// TwinCAT 3 PLC project Untitled1
// ProgramVersion: 3.1.4023.0
// libraries:
//   Motion, * (Ljmu)
//   SafetyMonitoring, * (Ljmu)
//   Tc2_ControllerToolbox, * (Beckhoff Automation GmbH)
//   Tc2_IoFunctions, * (Beckhoff Automation GmbH)
//   Tc2_MC2, * (Beckhoff Automation GmbH)
//   Tc2_MC2_Drive, * (Beckhoff Automation GmbH)
//   Tc2_NC, * (Beckhoff Automation GmbH)
//   Tc2_Standard, * (Beckhoff Automation GmbH)
//   Tc2_System, * (Beckhoff Automation GmbH)
//   Tc2_Utilities, * (Beckhoff Automation GmbH)
//   Tc3_EventLogger, * (Beckhoff Automation GmbH)
//   Tc3_IotBase, * (Beckhoff Automation GmbH)
//   Tc3_Module, * (Beckhoff Automation GmbH)
// project tree:
//   DUTs/ AGPowerStatus.TcDUT, Instrument.TcDUT, LinearPositions.TcDUT, RotationStates.TcDUT, LinearStates.TcDUT, st_EL1918Inputs.TcDUT, st_EL2904Outputs.TcDUT, ST_SafeEL1918Status.TcDUT, st_SafeEL2904Status.TcDUT
//   GVLs/ MovementPositions.TcGVL
//   POUs/ EverestMC.TcPOU, fbAGPowerStatus.TcPOU, fbEthercatStateMachine.TcPOU, fbSafetyStateAndDiagDecode.TcPOU, fbStateMachineManager.TcPOU, FB_SafeInfoState.TcPOU, IDXMotor.TcPOU, I_Motor.TcIO, MAIN.TcPOU, PlcTask.TcTTO, fSafetyStateAndDiagDecode.TcPOU, TestMode.TcPOU
// real-time tasks:
//   TASK PlcTask: cycle T#10ms, priority 20, ADS port 350
// motion (NC):
//   TASK NC-Task 1 SAF: cycle T#2ms, priority 4, ADS port 501
//   TASK NC-Task 1 SVB: cycle T#10ms, priority 8, ADS port 511
//   AXIS Linear (id 1)
//     Dynamic: AccelerationMaximum=12000, DecelerationMaximum=12000, Acceleration=1000, Deceleration=1000, Jerk=5000, DelayTime=0.006
//     Velo: RefSearch=10, RefSync=10, SlowManual=20, FastManual=200, Fast=250, Maximum=300
//     PositionAreaControl: Range=1
//     MotionControl: Enable=true, Range=0.005, Time=0.1
//     TargetPosControl: Range=0.1, Time=1
//     PEHControl: Enable=true
//     OtherSettings: AllowMotionCmdToSlave=true
//     encoder EncType=19
//       EncPara: ScaleFactorNumerator=0.0012207031, MaxCount=#xffffffff
//         SoftEndMinControl: Enable=true, Range=-10
//         SoftEndMaxControl: Enable=true, Range=500
//         ActPosCorrection: Enable=true
//         Inc: RefPosition=510, RefSoftSyncMask=#x0000ffff, HomingSensorSource=1
//     drive DrvType=16
//       DrvPara: MaxCount=#xffffffff, DriveControlDWord=#x00020000
//         Analog: VeloReferenz=250, TorqueSetpointScale=10, ScaleFactorActTorque=0.1
//         TimeComp: TaskDelayCycles=1
//     controller CtrType=1
//       CtrPara: PriorControlFactor=1
//         PosDiffControl: Enable=false
//         Observer: BandWidth=20
//   AXIS Rotation (id 2)
//     General: UnitName=°
//     Dynamic: AccelerationMaximum=1500, DecelerationMaximum=1500, Acceleration=100, Deceleration=100, Jerk=100
//     Velo: RefSearch=20, RefSync=4, SlowManual=10, FastManual=60, Fast=70, Maximum=90
//     PositionAreaControl: Range=1
//     MotionControl: Range=0.01
//     TargetPosControl: Range=0.1, Time=0.5
//     PEHControl: Enable=true
//     OtherSettings: AllowMotionCmdToSlave=true, PulseDistancePos=1, PulseDistanceNeg=1
//     encoder EncType=19
//       EncPara: ScaleFactorNumerator=0.001, MaxCount=#xffffffff
//         SoftEndMinControl: Enable=true, Range=-165
//         SoftEndMaxControl: Enable=true, Range=165
//         Inc: RefSearchInverse=true, RefSyncInverse=false, RefMode=1, HomingSensorSource=1
//     drive DrvType=16
//       DrvPara: MaxCount=#xffffffff, DriveControlDWord=#x00020000
//         Analog: VeloReferenz=80, TorqueSetpointScale=10, ScaleFactorActTorque=0.1
//         TimeComp: TaskDelayCycles=1
//     controller CtrType=1
//       CtrPara: PriorControlFactor=1
//         Observer: BandWidth=20
//   AXIS Linear Encoder (id 3)
//     OtherSettings: AllowMotionCmdToSlave=true
//     encoder EncType=4
//       EncPara: MaxCount=#x0000ffff
//         Inc: RefSoftSyncMask=#x0000ffff
//     drive DrvType=5
//       Analog: TorqueSetpointScale=10, ScaleFactorActTorque=0.1
//       TimeComp: TaskDelayCycles=1
//     controller CtrType=1
//       CtrPara: PriorControlFactor=1
//         Observer: BandWidth=20
//   AXIS Force (id 4)
//     General: UnitName=N
//     OtherSettings: AllowMotionCmdToSlave=true
//     encoder EncType=7
//       EncPara: ScaleFactorNumerator=2500, ScaleFactorDenominator=32768, Offset=-45, EncMode=1, MaxCount=#x0000ffff, ReferenceSystem=1
//         ActPosCorrection: Time=45
//     drive DrvType=5
//       Analog: TorqueSetpointScale=10, ScaleFactorActTorque=0.1
//       TimeComp: TaskDelayCycles=1
//     controller CtrType=1
//       CtrPara: PriorControlFactor=1
//         PosDiffControl: Enable=false
//         Observer: BandWidth=20
// I/O:
//   DEVICE Device 2 (EtherCAT), AmsNetId 5.119.202.92.3.1
//     Term 4 (EK1200) [EK1200-5000 EtherCAT Power supply (2A E-Bus)]
//       Term 6 (EL1918) [EL1918, 8Ch. Safety Input 24V, TwinSAFE]
//         modules: Module 2 (FSLOGIC)
//       Term 12 (EK1110) [EK1110 EtherCAT extension]
//     Drive 4 (IDX)
//     Box 18 (EP2338-0001) [EP2338-0001 8 Ch. Dig. Input/Output 24V, 0,5A, M8]
//     Box 19 (EP1957-0022) [EP1957, 8Ch. Safety Input 24V, 4Ch. Safety Output 24V, 0.5A, TwinSAFE]
//       modules: Module 1 (FSOE), Module 2 (FSOUT), Module 3 (DEVICEIO), Module 4 (FSLOGIC)
//     Term 21 (EK1100-0008) [EK1100-0008 EtherCAT Coupler M8 (2A E-Bus)]
//       Term 23 (EL5101) [EL5101 1Ch. Inc. Encoder 5V]
//       Term 24 (EL1918) [EL1918, 8Ch. Safety Input 24V, TwinSAFE]
//         modules: Module 1 (FSOE), Module 2 (FSLOGIC)
//       Term 25 (EL1004) [EL1004 4Ch. Dig. Input 24V, 3ms]
//       Term 26 (EL2904) [EL2904, 4 Ch. Safety Output 24V, 0.5A, TwinSAFE]
//         modules: Module 1 (FSOES), Module 2 (DO)
//       Term 16 (EL2002) [EL2002 2Ch. Dig. Output 24V, 0.5A]
//       Term 28 (EL3174-0042) [EL3174-0042 4Ch. Ana. Input +/-30V, +/-60V 16 Bit, Isolated Channels]
//       Term 20 (EL3314-0002) [EL3314-0002 4Ch. Ana Input Thermocouple (TC), Isolated Channels]
//       Term 18 (EL9011) [EL9011 End Terminal]
//     Drive 29 (EVS-XCR-E) [EVS-XCR-E]
// variable links:
//   Device 2 (EtherCAT) <-> Device 2 (EtherCAT)/Term 21 (EK1100-0008)/Term 24 (EL1918)
//     Term 4 (EK1200)/Term 6 (EL1918)/ConnectionInputs/TwinSafeGroup1.Term 24 (EL1918) - Module 1 (FSOE)_24 TxPDO <-> Module 1 (FSOE)/FSoE Outputs/FSOE
//     Term 4 (EK1200)/Term 6 (EL1918)/ConnectionOutputs/TwinSafeGroup1.Term 24 (EL1918) - Module 1 (FSOE)_24 RxPDO <-> Module 1 (FSOE)/FSoE Inputs/FSOE
//   Device 2 (EtherCAT) <-> Device 2 (EtherCAT)/Term 21 (EK1100-0008)/Term 26 (EL2904)
//     Term 4 (EK1200)/Term 6 (EL1918)/ConnectionInputs/TwinSafeGroup1.Term 26 (EL2904) - Module 1 (FSOES)_25 TxPDO <-> Module 1 (FSOES)/RxPDO/FSOE
//     Term 4 (EK1200)/Term 6 (EL1918)/ConnectionOutputs/TwinSafeGroup1.Term 26 (EL2904) - Module 1 (FSOES)_25 RxPDO <-> Module 1 (FSOES)/TxPDO/FSOE
//   NC-Task 1 SAF/Axes/Linear <-> Device 2 (EtherCAT)/Box 18 (EP2338-0001)
//     Drive/Inputs/In/nState8 <-> Channel 1/Input
//   NC-Task 1 SAF/Axes/Linear <-> Device 2 (EtherCAT)/Drive 4 (IDX)
//     Drive/Inputs/In/nDataIn3[0] <-> Module 1 (CSP Mode)/CSP Inputs/Torque actual value
//     Drive/Inputs/In/nDcOutputTime <-> InfoData/DcOutputShift
//     Drive/Inputs/In/nState1 <-> Module 1 (CSP Mode)/CSP Inputs/Statusword
//     Drive/Inputs/In/nState2 <-> Module 1 (CSP Mode)/CSP Inputs/Statusword @bit 8
//     Drive/Inputs/In/nState4 @bit 1 <-> WcState/InputToggle
//     Drive/Inputs/In/nState4 <-> WcState/WcStateIn
//     Drive/Inputs/In/nState5 <-> Module 1 (CSP Mode)/CSP Inputs/Mode of operation display
//     Drive/Outputs/Out/nCtrl1 <-> Module 1 (CSP Mode)/CSP Outputs/Controlword
//     Drive/Outputs/Out/nCtrl2 <-> Module 1 (CSP Mode)/CSP Outputs/Controlword @bit 8
//     Drive/Outputs/Out/nCtrl5 <-> Module 1 (CSP Mode)/CSP Outputs/Mode of operation
//     Drive/Outputs/Out/nDataOut1 <-> Module 1 (CSP Mode)/CSP Outputs/Target position
//     Drive/Outputs/Out/nDataOut3[0] <-> Module 1 (CSP Mode)/CSP Outputs/Torque offset
//     Enc/Inputs/In/nDataIn1 <-> Module 1 (CSP Mode)/CSP Inputs/Position actual value
//     Enc/Inputs/In/nDataIn7 <-> Module 1 (CSP Mode)/CSP Inputs/Velocity actual value
//     Enc/Inputs/In/nDcInputTime <-> InfoData/DcInputShift
//     Enc/Inputs/In/nState4 @bit 1 <-> WcState/InputToggle
//     Enc/Inputs/In/nState4 <-> WcState/WcStateIn
//   NC-Task 1 SAF/Axes/Linear Encoder <-> Device 2 (EtherCAT)/Term 21 (EK1100-0008)/Term 23 (EL5101)
//     Enc/Inputs/In/nDataIn1[0] <-> ENC Status compact/Counter value
//     Enc/Inputs/In/nDataIn2[0] <-> ENC Status compact/Latch value
//     Enc/Inputs/In/nState1 @bit 4 <-> ENC Status compact/Status/Counter overflow
//     Enc/Inputs/In/nState1 @bit 3 <-> ENC Status compact/Status/Counter underflow
//     Enc/Inputs/In/nState1 @bit 7 <-> ENC Status compact/Status/Extrapolation stall
//     Enc/Inputs/In/nState1 <-> ENC Status compact/Status/Latch C valid
//     Enc/Inputs/In/nState1 @bit 1 <-> ENC Status compact/Status/Latch extern valid
//     Enc/Inputs/In/nState1 @bit 6 <-> ENC Status compact/Status/Open circuit
//     Enc/Inputs/In/nState1 @bit 2 <-> ENC Status compact/Status/Set counter done
//     Enc/Inputs/In/nState1 @bit 5 <-> ENC Status compact/Status/Status of input status
//     Enc/Inputs/In/nState2 @bit 4 <-> ENC Status compact/Status/Status of extern latch
//     Enc/Inputs/In/nState2 <-> ENC Status compact/Status/Status of input A
//     Enc/Inputs/In/nState2 @bit 1 <-> ENC Status compact/Status/Status of input B
//     Enc/Inputs/In/nState2 @bit 2 <-> ENC Status compact/Status/Status of input C
//     Enc/Inputs/In/nState2 @bit 3 <-> ENC Status compact/Status/Status of input gate
//     Enc/Inputs/In/nState2 @bit 5 <-> ENC Status compact/Status/Sync error
//     Enc/Inputs/In/nState2 @bit 6 <-> ENC Status compact/Status/TxPDO State
//     Enc/Inputs/In/nState2 @bit 7 <-> ENC Status compact/Status/TxPDO Toggle
//     Enc/Inputs/In/nState4 @bit 1 <-> WcState/InputToggle
//     Enc/Inputs/In/nState4 <-> WcState/WcStateIn
//     Enc/Outputs/Out/nCtrl1 <-> ENC Control compact/Control/Enable latch C
//     Enc/Outputs/Out/nCtrl1 @bit 3 <-> ENC Control compact/Control/Enable latch extern on negative edge
//     Enc/Outputs/Out/nCtrl1 @bit 1 <-> ENC Control compact/Control/Enable latch extern on positive edge
//     Enc/Outputs/Out/nCtrl1 @bit 2 <-> ENC Control compact/Control/Set counter
//     Enc/Outputs/Out/nDataOut1[0] <-> ENC Control compact/Set counter value
//   NC-Task 1 SAF/Axes/Rotation <-> Device 2 (EtherCAT)/Drive 29 (EVS-XCR-E)
//     Drive/Inputs/In/nState1 <-> TPDO 1 mapping parameter/Status Word
//     Drive/Inputs/In/nState2 <-> TPDO 1 mapping parameter/Status Word @bit 8
//     Drive/Inputs/In/nState4 @bit 1 <-> WcState/InputToggle
//     Drive/Inputs/In/nState4 <-> WcState/WcStateIn
//     Drive/Inputs/In/nState5 <-> TPDO 1 mapping parameter/Operation mode display
//     Drive/Inputs/In/nState8 <-> TPDO 1 mapping parameter/Digital inputs value
//     Drive/Outputs/Out/nCtrl1 <-> RPDO 1 mapping parameter/Control Word
//     Drive/Outputs/Out/nCtrl2 <-> RPDO 1 mapping parameter/Control Word @bit 8
//     Drive/Outputs/Out/nCtrl5 <-> RPDO 1 mapping parameter/Operation mode
//     Drive/Outputs/Out/nDataOut1 <-> RPDO 1 mapping parameter/Position set-point
//     Drive/Outputs/Out/nDataOut2 <-> RPDO 1 mapping parameter/Velocity set-point
//     Enc/Inputs/In/nDataIn1 <-> TPDO 1 mapping parameter/Actual position
//     Enc/Inputs/In/nDataIn7 <-> TPDO 1 mapping parameter/Actual velocity
//     Enc/Inputs/In/nState4 @bit 1 <-> WcState/InputToggle
//     Enc/Inputs/In/nState4 <-> WcState/WcStateIn
//   Untitled1/Untitled1 Instance <-> Device 2 (EtherCAT)/Term 21 (EK1100-0008)/Term 16 (EL2002)
//     PlcTask Outputs/MAIN.LinearBrake <-> Channel 1/Output
//   Untitled1/Untitled1 Instance <-> Device 2 (EtherCAT)/Term 21 (EK1100-0008)/Term 24 (EL1918)
//     PlcTask Inputs/MAIN.AGSafeInputs.InputState <-> InfoData/State
//     PlcTask Inputs/MAIN.AGSafeInputs.InputWcState/InputToggle <-> WcState/InputToggle
//     PlcTask Inputs/MAIN.AGSafeInputs.InputWcState/WcState <-> WcState/WcStateIn
//   Untitled1/Untitled1 Instance <-> Device 2 (EtherCAT)/Term 21 (EK1100-0008)/Term 25 (EL1004)
//     PlcTask Inputs/MAIN.fbAGPowerStatus.AGPowerOk_1 <-> Channel 3/Input
//     PlcTask Inputs/MAIN.fbAGPowerStatus.AGPowerOk_2 <-> Channel 4/Input
//     PlcTask Inputs/MAIN.fbAGPowerStatus.MotorPowerOk_1 <-> Channel 1/Input
//     PlcTask Inputs/MAIN.fbAGPowerStatus.MotorPowerOk_2 <-> Channel 2/Input
//     PlcTask Inputs/MAIN.fbDigitalInputMonitor.InputState <-> InfoData/State
//     PlcTask Inputs/MAIN.fbDigitalInputMonitor.InputWcState/WcState <-> WcState/WcState
//   Untitled1/Untitled1 Instance <-> Device 2 (EtherCAT)/Term 21 (EK1100-0008)/Term 26 (EL2904)
//     PlcTask Inputs/MAIN.AGSafeOutputs.InputState <-> InfoData/State
//     PlcTask Inputs/MAIN.AGSafeOutputs.InputWcState/InputToggle <-> WcState/InputToggle
//     PlcTask Inputs/MAIN.AGSafeOutputs.InputWcState/WcState <-> WcState/WcStateIn
//   Untitled1/Untitled1 Instance <-> Device 2 (EtherCAT)/Term 21 (EK1100-0008)/Term 28 (EL3174-0042)
//     PlcTask Inputs/MAIN.LinearBrakeRawData <-> AI Standard Channel 3/Value
//     PlcTask Inputs/MAIN.fbAGPowerStatus.AGPowerRaw <-> AI Standard Channel 1/Value
//     PlcTask Inputs/MAIN.fbAGPowerStatus.DataInvalid <-> WcState/WcState
//     PlcTask Inputs/MAIN.fbAGPowerStatus.MotorPowerRaw <-> AI Standard Channel 2/Value
//   Untitled1/Untitled1 Instance <-> Device 2 (EtherCAT)/Term 4 (EK1200)/Term 6 (EL1918)
//     PlcTask Inputs/MAIN.AGEstop.EstopFBStateIn <-> Function Block Info Data/TwinSafeGroup1.Network1.AGBoxEstop Info Data/State
//     PlcTask Inputs/MAIN.AGEstop.bitStEstopFBDiag <-> Function Block Info Data/TwinSafeGroup1.Network1.AGBoxEstop Info Data/Diag
//     PlcTask Inputs/MAIN.AGSafeInputs.SafetyDiagnosis <-> Connection Info Data/TwinSafeGroup1.Term 24 (EL1918) - Module 1 (FSOE)_24 Info Data/Diag
//     PlcTask Inputs/MAIN.AGSafeInputs.SafetyState <-> Connection Info Data/TwinSafeGroup1.Term 24 (EL1918) - Module 1 (FSOE)_24 Info Data/State
//     PlcTask Inputs/MAIN.AGSafeOutputs.Outputs/Output{1..4} <-> Connection Info Data/TwinSafeGroup1.Term 26 (EL2904) - Module 1 (FSOES)_25 Info Data/Output Safe Data OutputChannel{1..4}  (4 links)
//     PlcTask Inputs/MAIN.AGSafeOutputs.SafetyDiagnosis <-> Connection Info Data/TwinSafeGroup1.Term 26 (EL2904) - Module 1 (FSOES)_25 Info Data/Diag
//     PlcTask Inputs/MAIN.AGSafeOutputs.SafetyState <-> Connection Info Data/TwinSafeGroup1.Term 26 (EL2904) - Module 1 (FSOES)_25 Info Data/State
//     PlcTask Inputs/MAIN.OffMountEstop.EstopFBStateIn <-> Function Block Info Data/TwinSafeGroup1.Network1.OffMountEstop Info Data/State
//     PlcTask Inputs/MAIN.OffMountEstop.bitStEstopFBDiag <-> Function Block Info Data/TwinSafeGroup1.Network1.OffMountEstop Info Data/Diag
//     PlcTask Inputs/MAIN.SafetySystem.GlobalEstopStatus <-> StandardInputs/TwinSafeGroup1.EstopToPLC_7
//     PlcTask Inputs/MAIN.SafetySystem.eSafetyGroupDiagnosis <-> TwinSAFE Group Info Data/TwinSafeGroup1 Info Data/Diag
//     PlcTask Inputs/MAIN.SafetySystem.eSafetyGroupState <-> TwinSAFE Group Info Data/TwinSafeGroup1 Info Data/State
//     PlcTask Inputs/MAIN.fbSafetyMasterMonitor.InputState <-> InfoData/State
//     PlcTask Inputs/MAIN.fbSafetyMasterMonitor.InputWcState/InputToggle <-> WcState/InputToggle
//     PlcTask Inputs/MAIN.fbSafetyMasterMonitor.InputWcState/WcState <-> WcState/WcStateIn
//     PlcTask Outputs/MAIN.SafetySystem.ErrAck <-> StandardOutputs/TwinSafeGroup1.ErrorAcknowledgement_1
//     PlcTask Outputs/MAIN.SafetySystem.Run <-> StandardOutputs/TwinSafeGroup1.Run_2
//   Untitled1/Untitled1 Instance <-> NC-Task 1 SAF/Axes/Force
//     PlcTask Inputs/MAIN.Force.NcToPlc <-> Outputs/ToPlc
//     PlcTask Outputs/MAIN.Force.PlcToNc <-> Inputs/FromPlc
//   Untitled1/Untitled1 Instance <-> NC-Task 1 SAF/Axes/Linear
//     PlcTask Inputs/MAIN.LinearMotor.Axis.NcToPlc <-> Outputs/ToPlc
//     PlcTask Outputs/MAIN.LinearMotor.Axis.PlcToNc <-> Inputs/FromPlc
//   Untitled1/Untitled1 Instance <-> NC-Task 1 SAF/Axes/Linear Encoder
//     PlcTask Inputs/MAIN.LinearEncoder.NcToPlc <-> Outputs/ToPlc
//     PlcTask Outputs/MAIN.LinearEncoder.PlcToNc <-> Inputs/FromPlc
//   Untitled1/Untitled1 Instance <-> NC-Task 1 SAF/Axes/Rotation
//     PlcTask Inputs/MAIN.fbEverest.Axis.NcToPlc <-> Outputs/ToPlc
//     PlcTask Outputs/MAIN.fbEverest.Axis.PlcToNc <-> Inputs/FromPlc

CONFIGURATION Untitled1
    RESOURCE PLC ON TwinCAT3
        TASK PlcTask(INTERVAL := T#10ms, PRIORITY := 20);
        PROGRAM MAIN WITH PlcTask : MAIN;
    END_RESOURCE
END_CONFIGURATION

// ---- DUTs/AGPowerStatus.TcDUT
TYPE AGPowerStatus :
STRUCT
	MotorPowerRaw AT%I* :INT;
	MotorPowerV :REAL;
	AGPowerRaw AT%I* :INT;
	AGPowerV:REAL;
	MotorPowerOk_1 AT%I* :BOOL;
	MotorPowerOk_2 AT%I* :BOOL;
	AGPowerOk_1 AT%I*:BOOL;
	AGPowerOk_2 AT%I*:BOOL;
	AllPSUOK :BOOL;
	
END_STRUCT
END_TYPE

// ---- DUTs/Instrument.TcDUT
TYPE Instrument :
STRUCT
	Name		:STRING;
	Rotation	:LREAL	:=1000;
	Linear		:LREAL	:=0;
	Enabled 	:BOOL	:=TRUE;

END_STRUCT
END_TYPE

// ---- DUTs/LinearPositions.TcDUT
TYPE LinearPositions :
STRUCT
	Deployed :LREAL:=100;
	Stowed :LREAL:=500;
	maintenance :LREAL:=0;
	
END_STRUCT
END_TYPE

// ---- DUTs/RotationStates.TcDUT
{attribute 'qualified_only'}
{attribute 'strict'}
TYPE RotationStates :
(
	Initialising,
	Start_Homing,
	Homing,
	Idle,
	Start_Move,
	Moving,
	Error
);
END_TYPE

// ---- DUTs/LinearStates.TcDUT
{attribute 'qualified_only'}
{attribute 'strict'}
{attribute 'to_string'}
TYPE LinearStates :
(
	Initialising,
	Start_Homing,
	Homing,
	Idle,
	Start_Move,
	Moving,
	Error
);
END_TYPE

// ---- DUTs/st_EL1918Inputs.TcDUT
TYPE st_EL1918Inputs :
STRUCT
	Input1 :BIT;
	Input1Err :BIT;
	Input2 :BIT;
	Input2Err :BIT;
	Input3 :BIT;
	Input3Err :BIT;
	Input4 :BIT;
	Input4Err :BIT;
	Input5 :BIT;
	Input5Err :BIT;
	Input6 :BIT;
	Input6Err :BIT;
	Input7 :BIT;
	Input7Err :BIT;
	Input8 :BIT;
	Input8Err :BIT;
	
END_STRUCT
END_TYPE

// ---- DUTs/st_EL2904Outputs.TcDUT
TYPE st_EL2904Outputs :
STRUCT
	Output1 :BIT;
	Output2 :BIT;
	Output3 :BIT;
	Output4 :BIT;
	
END_STRUCT
END_TYPE

// ---- DUTs/ST_SafeEL1918Status.TcDUT
TYPE ST_SafeEL1918Status :
STRUCT
	State AT%I* :USINT;
	Diag AT%I* :USINT;
	Status :st_SafetyStatus;
	Inputs AT%I* :st_EL1918Inputs;
END_STRUCT
END_TYPE

// ---- DUTs/st_SafeEL2904Status.TcDUT
TYPE st_SafeEL2904Status :
STRUCT
	State AT%I* :USINT;
	Diag AT%I* :USINT;
	Status :st_SafetyStatus;
	Outputs AT%I* :st_EL2904Outputs;
END_STRUCT
END_TYPE

// ---- GVLs/MovementPositions.TcGVL
{attribute 'qualified_only'}
VAR_GLOBAL
	//units mm
linearpos	:linearPositions;
	//units degrees
	InstrumentPositions	:ARRAY [0..7] OF Instrument := [(Name:='raptor',Rotation:=1000, Linear :=100,Enabled :=TRUE),
														(Name:='IRCam',Rotation:=2000, Linear :=100,Enabled :=TRUE),
														(Name:='Spec',Rotation:=3000, Linear :=100,Enabled :=TRUE),
														(Name:='Chimera',Rotation:=4000, Linear :=100,Enabled :=TRUE),
														(Name:='Dave',Rotation:=5000, Linear :=100,Enabled :=TRUE),
														(Name:='Galileo',Rotation:=6000, Linear :=100,Enabled :=TRUE),
														(Name:='CARIBOU',Rotation:=3000, Linear :=500,Enabled :=TRUE)];

	
END_VAR

// ---- POUs/I_Motor.TcIO
INTERFACE I_Motor

METHOD PUBLIC Enable : BOOL
VAR_INPUT
EnableMotor :BOOL;
END_VAR
END_METHOD

METHOD PUBLIC Home : BOOL
VAR_IN_OUT
	Execute:BOOL;
END_VAR
END_METHOD

METHOD Homed : BOOL
VAR_INPUT
END_VAR
END_METHOD

METHOD MoveRelative : BOOL
VAR_INPUT
	Distance: LREAL;
	Velocity: LREAL;	
END_VAR
VAR_IN_OUT
	Execute: BOOL;
END_VAR
END_METHOD

METHOD MoveTo : BOOL
VAR_INPUT
	Position: LREAL;
	Velocity: LREAL;	
END_VAR

VAR_OUTPUT
	State :e_MCState;
	Target : LREAL;
END_VAR

VAR_IN_OUT
		Execute: BOOL;
END_VAR
END_METHOD

METHOD Position : LREAL
VAR_INPUT
END_VAR
END_METHOD

METHOD Reset : BOOL
VAR_IN_OUT
	ResetAxis:BOOL;
	//IDXControlByte1 :USINT;
END_VAR
END_METHOD

METHOD PUBLIC Status : ST_AxisStatus
VAR_INPUT
END_VAR
END_METHOD

END_INTERFACE

// ---- POUs/MAIN.TcPOU
PROGRAM MAIN
VAR CONSTANT 

	SafetyModuleArraySize :UINT:=1;
	EstopArraySize :UINT := 1;
END_VAR
VAR
	LinearErrorArray : ST_IDXError;
	LinearMotor :FB_Motion(AxisNameIn := 'M3 Linear');
	LinearBrake AT%Q*:BOOL;
	fbIDXError: FB_IDXError(AxisNameIn := 'M3 Linear');


	SafetySystem : FB_SafetySystemMonitor;
	AGSafeInputs : FB_EL1918Monitor(Namein:='AGSafeInputs',ElectricalRefin:='K7',Addressin:=1008);
	AGSafeOutputs : FB_EL2904Monitor(NameIn:='AGSafeOutputs',ElectricalRefIn:='K8',AddressIn:=1010);
	AGEstop: FB_SafetyEstopMonitor(NameIn:='A&G Box');
	OffMountEstop :FB_SafetyEstopMonitor(NameIn:='Off Mount');

	fbDigitalInputMonitor : FB_EthercatModuleMonitor(NameIn:='AGDigitalInput',ElectricalRefIn:='K2',AddressIn:=1009);
	fbLinearMotorMonitor : FB_EthercatModuleMonitor(NameIn:='AGLinearMotorInput',ElectricalRefIn:='M2',AddressIn:=1003);
	fbSafetyMasterMonitor : FB_EthercatModuleMonitor(NameIn:='SafetyMaster',ElectricalRefIn:='K1',AddressIn:=1001);
	
		{attribute 'OPC.UA.DA' := '1'}
	{attribute 'OPC.UA.DA.Access' := '1'}
	{attribute 'OPC.UA.DA.StructuredType' := '0'}
	SafetyModuleStatus : ARRAY[0..SafetyModuleArraySize] OF ST_SafetyModule;
	fbsafetyModuleCollector :FB_SafetyModuleCollector;
	{attribute 'OPC.UA.DA' := '1'}
	{attribute 'OPC.UA.DA.Access' := '1'}
	{attribute 'OPC.UA.DA.StructuredType' := '0'}
	EstopArray : ARRAY [0..EstopArraySize] OF ST_EstopFB;
	fbEstopFBCollector : FB_EstopFBCollector;

	fbEverest :EverestMC();
	LinearEncoder: AXIS_REF;
	Force: AXIS_REF;
	fbIDXResetError : FB_IDXResetError(AxisNameIn := 'M3 Linear');
	ResetError :BOOL;
	GetUPSStatus : FB_GetUPSStatus;
	ReadUPSStatus:BOOL := TRUE;
	
	{attribute 'OPC.UA.DA' := '1'}
	{attribute 'OPC.UA.DA.Access' := '1'}
	{attribute 'OPC.UA.DA.StructuredType' := '0'}
	fbAGPowerStatus : fbAGPowerStatus;

	
	{attribute 'OPC.UA.DA' := '1'}
	{attribute 'OPC.UA.DA.Access' := '1'}
	{attribute 'OPC.UA.DA.StructuredType' := '0'}
	UPSStatus: ST_UPSStatus;
	UPSStatusValid:BOOL;
	
	Instruments :ARRAY[0..4] OF Instrument ;
	{attribute 'OPC.UA.DA' := '1'}
	DemoMode: BOOL;
	CurrentInstrument:INT;
	Change_Inst :TON:= (PT:=T#10S,IN:=FALSE);
	CurrentInstName:STRING;
	
	
	
	ForceAvg : FB_CTRL_MOVING_AVERAGE;
	ForceAvgArray: ARRAY[0..100] OF LREAL;
	ForceAvgParas : ST_CTRL_MOVING_AVERAGE_PARAMS := (
tCtrlCycleTime:= T#100MS,
tTaskCycleTime:= T#10MS,
nSamplesToFilter:=100,
pWorkArray_ADR:= ADR(ForceAvgArray),
nWorkArray_SIZEOF:= 800);


	
	{attribute 'OPC.UA.DA' := '1'}
	IdxEnable:BOOL;
	{attribute 'OPC.UA.DA' := '1'}
	EveEnable:BOOL;

	{attribute 'OPC.UA.DA' := '1'}
	{attribute 'OPC.UA.DA.Access' := '1'}
	Estop: BOOL;
	RotationHome :BOOL:=FALSE;
	LinearResetAxis :BOOL:=FALSE;
	LinearResetNC	:BOOL := FALSE;
	RotationresetAxis :BOOL:=FALSE;
	FBLInearEncHome :MC_Home;
LinearEncHome:BOOL;
LinearHomePosition:LREAL;



LinearBrakeRawData AT %I* :INT;
LinearBrakePressure		:LREAL; //bar
LinearBrakeMinOperatingPressure:LREAL:= 5.0; //bar
LinearBrakeUnderPressure :BOOL;
fbLinearBrakePressureScale :FB_CTRL_SCALE;
LinearBrakeScaleParams : ST_CTRL_SCALE_PARAMS:=(
	fInMax:=10000.0,//mv
	fInMin:=0.0,//mv
	fOutMax:=10.0,//bar
	fOutMin:= 0.0,//bar
	tCtrlCycleTime:=T#500MS,
	tTaskCycleTime:= T#10MS);
BrakeUnderPressureTimer :ton := (PT:= T#250MS); // timer prevents small dips of pressure during valves opens to disable motor

	
	{attribute 'OPC.UA.DA' := '1'}
	LinearAxisState: LinearStates; (*~ (OPC:1:linear axis status ) *)
	{attribute 'OPC.UA.DA' := '1'}
	LinearCommandedPosition:LREAL:=400;

	LinearMove:BOOL;
	LinearMoveState: e_MCState;
	{attribute 'OPC.UA.DA' := '1'}
	LinearErrorACK:BOOL:=FALSE;
	{attribute 'OPC.UA.DA' := '1'}
	LinearMovementSpeed:LREAL:=50;
		{attribute 'OPC.UA.DA' := '1'}
	{attribute 'OPC.UA.DA.Access' := '1'}
	{attribute 'OPC.UA.DA.StructuredType' := '0'}
	LinearStatus :ST_AxisStatus;
	{attribute 'OPC.UA.DA' := '1'}
	{attribute 'OPC.UA.DA.Access' := '1'}
{attribute 'OPC.UA.DA.Description' := 'Position of Linear Stage'}
	LinearPosition  : LREAL;
	

	
	
	RotationStatus: ST_AxisStatus;
	{attribute 'OPC.UA.DA' := '1'}
	RotationPosition: LREAL;
	LinearHome: BOOL;
	{attribute 'OPC.UA.DA' := '1'}
	RotationAxisState: RotationStates;
	{attribute 'OPC.UA.DA' := '1'}
	RotationCommandedPosition: LREAL:=60;
	{attribute 'OPC.UA.DA' := '1'}
	RotationMovementSpeed: LREAL:=20;
	RotationMove: BOOL;
	HomingBusy: BOOL;
	
	



	RotationErrorACK: BOOL;
	SafetyMasterStatus: ST_EthercatStatus;

END_VAR


	
//standard module monitoring 
fbDigitalInputMonitor();
fbLinearMotorMonitor();
fbSafetyMasterMonitor();
fbSafetyMasterMonitor.GetEthercatStatus(stEthercatStatusOut=>SafetyMasterStatus);

SafetySystem.SetMasterStatus(StEthercatStatusIn:=SafetyMasterStatus);
SafetySystem();
Estop := SafetySystem.GetGlobalEstopStatus(); // true means system running 
//SafetyModules 
AGSafeInputs();
fbsafetyModuleCollector.GetSafetyStatus(StModuleArrayInOut:= SafetyModuleStatus,
 										ModuleArraySizeIn:=SafetyModuleArraySize,
										SafetyModuleRefIn:= AGSafeInputs,
										ModuleIndexIn:=0);
AGSafeOutputs();
fbsafetyModuleCollector.GetSafetyStatus(StModuleArrayInOut:= SafetyModuleStatus,
 										ModuleArraySizeIn:=SafetyModuleArraySize,
										SafetyModuleRefIn:= AGSafeOutputs,
										ModuleIndexIn:=1);
 //EstopGroups 
AGEstop();
OffMountEstop();
fbEstopFBCollector.GetEstopData(SafetyEstopRefIn:= AGEstop,
								stEstopArrayInOut:= EstopArray,
								EstopArraySizeIn:= EstopArraySize,
								EstopIndexIn:=0);
fbEstopFBCollector.GetEstopData(SafetyEstopRefIn:= OffMountEstop,
								stEstopArrayInOut:= EstopArray,
								EstopArraySizeIn:= EstopArraySize,
								EstopIndexIn:=1);
fbEstopFBCollector.MasterDataValid(DataValidIn:= SafetyMasterStatus.DataValid);
// DataCollectors 
fbsafetyModuleCollector(stModuleArrayInOut:= SafetyModuleStatus, ModuleArraySizeIn:=SafetyModuleArraySize);
fbEstopFBCollector(stEstopArrayInOut:= EstopArray, EstopArraySizeIn:= EstopArraySize);


//fbIDXError(Axis := fbIDX70.axis);
//fbIDXError.GetErrorStructure(StIDXErrorOut=> stIDXError);


LinearEncoder.ReadStatus();
Force.ReadStatus();

LinearMotor();
fbEverest();
fbAGPowerStatus();



// AND IdxEnable AND EveEnable
IF DemoMode  AND Change_Inst.Q  THEN
	CurrentInstrument:= (CurrentInstrument+1) MOD 4;
	Change_Inst(IN :=FALSE);
	LinearCommandedPosition:= (CurrentInstrument*75);
	RotationCommandedPosition:= (CurrentInstrument*60)-120;
	CurrentInstName := Instruments[CurrentInstrument].Name;
ELSIF  NOT DemoMode THEN
	CurrentInstName :=' None Selected ';
ELSE 
	Change_Inst(IN :=TRUE);

	
END_IF



ForceAvg(
 fIn:= Force.NcToPlc.ActPos,
stParams:= ForceAvgParas,
eMode:= E_CTRL_MODE.eCTRL_MODE_ACTIVE);
	

	FBLinearEncHome(
	Axis:=LinearEncoder,
	Execute:=LinearEncHome,
	Position:=LinearHomePosition,
	HomingMode:=MC_Direct);
	


	
GetUPSStatus(sNetId:='',
	Nport:=0,  (* 0 = Windows UPS service / Windows Battery driver  *)
	bEnable:= ReadUPSStatus,
	bValid=>UPSStatusValid,
	stStatus=> UPSStatus);



fbIDXError(Axis:=LinearMotor.Axis);
fbIDXError.GetErrorStructure(StIDXErrorOut=> LinearErrorArray);
//fbMotionEventSender.MotorError(stIDXError:=LinearErrorArray);

fbIDXResetError(Execute:= LinearresetAxis,Axis:=LinearMotor.Axis); 
fbLinearBrakePressureScale(
	fIn:= LinearBrakeRawData,
	stParams:= LinearBrakeScaleParams,
	fOut=> LinearBrakePressure);

// Estop is active low 
IF NOT Estop THEN  //Estop check
	IdxEnable:=FALSE;
	EveEnable:=FALSE;	
END_IF

IF LinearBrakePressure<LinearBrakeMinOperatingPressure THEN
	LinearBrakeUnderPressure := TRUE;
ELSE 
	LinearBrakeUnderPressure := FALSE;
END_IF
BrakeUnderPressureTimer(IN:= LinearBrakeUnderPressure);

IF BrakeUnderPressureTimer.Q THEN
	IdxEnable:=FALSE;
END_IF
LinearBrake := IdxEnable;// brake disabled when motor online 
LinearMotor.Estop(Execute:= NOT Estop );



LinearMotor.Enable(Execute:= IdxEnable);
LinearMotor.Reset(Execute := LinearResetNC);
HomingBusy:= LinearMotor.Home(Execute:= LinearHome,HomePositionIn:= 510.0);
LinearMotor.GetCurrentPosition(PositionOut=> LinearPosition);
LinearMotor.GetStatus(AxisOut:= LinearStatus);

LinearMotor.MoveTo(
	Execute:= LinearMove,
	TargetPositionIn:= LinearCommandedPosition,
	VelocityIn := LinearMovementSpeed,
	eStateOut=> LinearMoveState);

IF LinearStatus.Error  THEN // put in error state if axis is in error 
	LinearAxisState:=LinearStates.Error;
ELSIF NOT IdxEnable THEN // if not in error or enabled 
		LinearAxisState:=LinearStates.Initialising;
		
END_IF

CASE(LinearAxisState) OF 
	
	LinearStates.Initialising:
		
		IF  LinearStatus.Operational AND LinearStatus.Homed THEN
			LinearAxisState:=LinearStates.Idle;	
		ELSIF LinearStatus.Operational THEN 
			LinearAxisState:=LinearStates.Start_Homing;
		END_IF
	
	LinearStates.Start_Homing:
		LinearHome:=TRUE;
		LinearAxisState:=LinearStates.Homing;

	LinearStates.Homing:
		IF LinearStatus.Homed AND NOT HomingBusy THEN
			LinearAxisState:=LinearStates.Idle;
		
		END_IF
	
	LinearStates.Idle:
		IF ABS(LinearCommandedPosition-LinearPosition)>0.01  THEN
			LinearAxisState:=LinearStates.Start_Move;
		ELSE
			LinearMove:=FALSE;
		END_IF
		
	LinearStates.Start_Move:
			LinearMove:=TRUE;
			LinearAxisState:=LinearStates.Moving; 
			
	LinearStates.Moving:
		IF LinearMoveState = e_MCState.Done THEN
			LinearAxisState:=LinearStates.Idle; 
			
		ELSIF LinearMoveState = e_MCState.Error THEN
			LinearAxisState:=LinearStates.Error; 
		END_IF
	
	LinearStates.Error:
	IdxEnable:=FALSE;
		IF LinearErrorACK THEN
			LinearResetAxis:=TRUE;
			LinearResetNC := TRUE;
			LinearErrorACK:=FALSE;
			LinearAxisState:= LinearStates.Initialising;
		END_IF

	
END_CASE


RotationStatus:= fbEverest.Status();
fbEverest.Enable(EnableMotor:= EveEnable);
fbEverest.Reset(resetAxis:=RotationresetAxis);
fbEverest.Home(Execute:=RotationHome);
RotationPosition := fbEverest.Position();
fbEverest.MoveTo(Position:=RotationCommandedPosition,Velocity:=RotationMovementSpeed,Execute:=RotationMove);

IF RotationStatus.Error THEN
	RotationAxisState:=RotationStates.Error;
ELSIF NOT EveEnable THEN
		RotationAxisState:=RotationStates.Initialising;
END_IF


CASE(RotationAxisState) OF 
	
	RotationStates.Initialising:
		
		IF  RotationStatus.Operational THEN
			RotationAxisState:=RotationStates.Start_Homing;
		END_IF
	
	RotationStates.Start_Homing:
	IF RotationStatus.Homed THEN
			RotationAxisState:=RotationStates.Idle;
		ELSE
			RotationHome:=TRUE;
			RotationAxisState:=RotationStates.Homing;
		END_IF
	

	RotationStates.Homing:
	IF RotationStatus.Homed THEN
			RotationAxisState:=RotationStates.Idle;
	END_IF
			
		
	
	RotationStates.Idle:
		IF ABS(RotationCommandedPosition-fbEverest.Axis.NcToPlc.SetPos)>0.01 THEN
			RotationAxisState:=RotationStates.Moving;
			RotationMove:=TRUE;
		ELSE 
			RotationMove:=FALSE;
		END_IF
		
			
	RotationStates.Moving:
		IF NOT RotationStatus.HasJob THEN
			RotationAxisState:=	RotationStates.Idle;
		END_IF
	
	RotationStates.Error:
		IF RotationErrorACK THEN
			RotationresetAxis:=TRUE;
			RotationErrorACK:=FALSE;
		END_IF
		
	
END_CASE

END_PROGRAM

// ---- POUs/EverestMC.TcPOU
FUNCTION_BLOCK EverestMC implements I_Motor
VAR_INPUT
	//
END_VAR
VAR_OUTPUT
END_VAR
VAR
	Axis: AXIS_REF;
	Enabled: BOOL := FALSE;
	Override: LREAL:=100;
	MotorError AT%I*	:WORD;
	MotorErrorSent : WORD;
	AxisErrorSent:UDINT;
	NCError : WORD;
	fbMessage : FB_TcMessage;
	EnableEventSent:BOOL:= TRUE;
	HomeEventSent:BOOL:=TRUE;
	MovementFinishedEventSent:BOOL;
    fbAxisMoveAbsolute: MC_MoveAbsolute;	
	fbMcHome: MC_Home;
	fbAxisPower: MC_Power;
	fbReset: MC_Reset;
	fbMoveRel : MC_MoveRelative;
	
END_VAR

Axis.ReadStatus();

IF NOT (MotorError = MotorErrorSent) THEN// Creates Event 
	MotorErrorSent:= MotorError;
	fbMessage.CreateEx(TC_Events.LinearMotor.IDXmotorError,0);
	fbMessage.ipArguments.Clear().AddDWord(MotorError);
	fbMessage.Send(0);
END_IF

IF NOT (Axis.NcToPlc.ErrorCode = AxisErrorSent) THEN// Creates Event 
	AxisErrorSent:= Axis.NcToPlc.ErrorCode;
	fbMessage.CreateEx(TC_Events.LinearMotor.AxisError,0);
	fbMessage.ipArguments.Clear().AddDWord(Axis.NcToPlc.ErrorCode);
	fbMessage.Send(0);
END_IF

METHOD Enable : BOOL
VAR_INPUT
	EnableMotor :BOOL;
END_VAR
	fbAxisPower( // use in idx class
    Axis:= Axis,
    Enable:= EnableMotor,
    Enable_Positive:= EnableMotor,
    Enable_Negative:= EnableMotor,
    Override:= Override,
	Status=>Enable,
	Error=>
);

IF EnableMotor = EnableEventSent THEN	
	EnableEventSent := NOT EnableEventSent;
IF EnableMotor THEN
	fbMessage.CreateEx(TC_Events.LinearMotor.Motor_enabled,0);
ELSE
	fbMessage.CreateEx(TC_Events.LinearMotor.Motor_disabled,0);
END_IF
//fbMessage.Send(0);
END_IF
END_METHOD

METHOD Estop : BOOL
VAR_INPUT
END_VAR
END_METHOD

METHOD PUBLIC Home : BOOL
VAR_IN_OUT
	Execute:BOOL;
END_VAR
VAR
	HomingDone:BOOL;
	HomingError:BOOL;
	HomingErrorID:UDINT;
END_VAR
// try changing limits to no error mode then home 


	fbMcHome(
	Axis:=Axis,
	Execute:=Execute,
	//Position:=510,
	HomingMode:=MC_DefaultHoming,
	Busy=>Home,
	Done=>HomingDone,
	Error=> HomingError,
	ErrorID=> HomingErrorID
);
	
IF Execute THEN
	HomeEventSent:= FALSE;
	fbMessage.CreateEx(TC_Events.LinearMotor.Homing,0);
	//fbMessage.Send(0);
	Execute:= FALSE;	
END_IF
IF HomingDone THEN
	fbMessage.CreateEx(TC_Events.LinearMotor.HomingComplete,0);
	//fbMessage.Send(0);
END_IF

IF HomingError THEN
	fbMessage.CreateEx(TC_Events.LinearMotor.HomingFailed,0);
	fbMessage.ipArguments.Clear().AddDWord(HomingErrorID);
	//fbMessage.Send(0);
END_IF
END_METHOD

METHOD PUBLIC Homed : BOOL
VAR_INPUT
END_VAR
Homed:=Axis.NcToPlc.StateDWord.1;
END_METHOD

METHOD MoveRelative : BOOL
VAR_INPUT
	Distance: LREAL;
	Velocity: LREAL;	
END_VAR
VAR_IN_OUT
	Execute: BOOL;
END_VAR
	fbMoveRel( // in idx class 
    Axis:= Axis,
    Execute:= Execute,
    Distance:= Distance,
    Velocity:= Velocity,);
	
		IF Execute THEN
	fbMessage.CreateEx(TC_Events.LinearMotor.RelativeMove,0);
	fbMessage.ipArguments.Clear();
	fbMessage.ipArguments.AddLReal(Distance);
	fbMessage.ipArguments.AddLReal(Velocity);
	//fbMessage.Send(0);
	Execute := FALSE;
END_IF

IF fbMoveRel.Done  THEN
	fbMessage.CreateEx(TC_Events.LinearMotor.MoveComplete,0);
	//fbMessage.Send(0);
	
END_IF
END_METHOD

METHOD PUBLIC MoveTo : BOOL
VAR_INPUT
	Position: LREAL;
	Velocity: LREAL;	
END_VAR

VAR_OUTPUT
	State:e_MCState;
	Target : LREAL;
END_VAR

VAR_IN_OUT
		Execute: BOOL;
END_VAR
 	fbAxisMoveAbsolute( // in idx class 
    Axis:= Axis,
    Execute:= Execute,
    Position:= Position,
    Velocity:= Velocity,);
	
	IF Execute THEN
	fbMessage.CreateEx(TC_Events.LinearMotor.MotorMove,0);
	fbMessage.ipArguments.Clear();
	fbMessage.ipArguments.AddLReal(Position);
	fbMessage.ipArguments.AddLReal(Velocity);
	//fbMessage.Send(0);
	Execute := FALSE;

END_IF

IF fbAxisMoveAbsolute.Done  THEN
	fbMessage.CreateEx(TC_Events.LinearMotor.MoveComplete,0);
	//fbMessage.Send(0);

	
END_IF
END_METHOD

METHOD Position : LREAL
VAR_INPUT
END_VAR
Position:= Axis.NcToPlc.ActPos;
END_METHOD

METHOD Reset : BOOL
VAR_IN_OUT
	ResetAxis:BOOL;
END_VAR
fbReset(
Axis:=Axis,
Execute:=ResetAxis,
Done =>Reset);

IF resetAxis THEN
//IDXControlByte1 := 16#80;// restop linear Motor
//MotorResetBit := 16#80;
fbMessage.CreateEx(TC_Events.LinearMotor.AxisReset,0);
//fbMessage.send(0);
resetAxis := FALSE;
END_IF
END_METHOD

METHOD PUBLIC Status : ST_AxisStatus
VAR_INPUT
END_VAR
Status := Axis.Status;
END_METHOD

END_FUNCTION_BLOCK

// ---- POUs/fbAGPowerStatus.TcPOU
FUNCTION_BLOCK fbAGPowerStatus
VAR
	//PowerStatus :AGPowerStatus;
	{attribute 'OPC.UA.DA' := '0'}
	MotorPowerRaw AT%I* :INT;
	MotorPowerV :REAL;
	{attribute 'OPC.UA.DA' := '0'}
	AGPowerRaw AT%I* :INT;
	AGPowerV:REAL;
	MotorPowerOk_1 AT%I* :BOOL;
	MotorPowerOk_2 AT%I* :BOOL;
	AGPowerOk_1 AT%I*:BOOL;
	AGPowerOk_2 AT%I*:BOOL;
	AllPSUOK :BOOL;
	AGPSUOK :BOOL;
	MOTORPSUOK:BOOL;
	{attribute 'OPC.UA.DA' := '0'}
	MotorPowerConversion:REAL :=128.4/65536.0 ;// 16 bit set to +-60 so 2^16/120 however extended range gives 7% more range 
	{attribute 'OPC.UA.DA' := '0'}
	AGPowerConversion:REAL :=64.2/65536.0;// set to +-30
	DataInvalid AT%I* :BOOL;
END_VAR

IF DataInvalid THEN
	AGPowerRaw := 0;
	MotorPowerRaw:=0;
END_IF

MotorPowerV := MotorPowerRaw*MotorPowerConversion;
AGPowerV := AGPowerRaw*AGPowerConversion;
MotorPSUOK := MotorPowerOk_1 AND MotorPowerOk_2 ;
AGPSUOK := AGPowerOk_1 AND AGPowerOk_2;
AllPSUOK := AGPSUOK AND MOTORPSUOK;

END_FUNCTION_BLOCK

// ---- POUs/fbEthercatStateMachine.TcPOU
FUNCTION_BLOCK fbEthercatStateMachine
VAR
	InputState AT%I*	:UINT;	
	WcState AT%I* :BOOL;
	InternalEtherCatState : st_EthercatState;
	
{attribute 'OPC.UA.DA' := '0'}	
	State :UINT;
		
{attribute 'OPC.UA.DA' := '0'}
	Error:UINT;
	
END_VAR

// table of states https://infosys.beckhoff.com/english.php?content=../content/1033/b110_ethercat_optioninterface/1984417163.html&id=
// uint is 16 bit final 4 bit are state first 12 are error 
State := InputState AND 16#000F;
Error := InputState AND 16#FFF0;
InternalEtherCatState.State:= UINT_TO_INT(State);
InternalEtherCatState.Error := UINT_TO_INT(Error);
InternalEtherCatState.DataInvalid := WcState;

METHOD FB_init : BOOL
VAR_INPUT
	bInitRetains : BOOL; // if TRUE, the retain variables are initialized (warm start / cold start)
	bInCopyCode : BOOL;  // if TRUE, the instance afterwards gets moved into the copy code (online change)
	EtherCatAddr : T_AmsNetID;
	nSlaveAddr : UINT;
END_VAR
InternalEtherCatState.nSlaveAddr:= nSlaveAddr;
InternalEtherCatState.EtherCatAddr := EtherCatAddr;
END_METHOD

METHOD GetState : BOOL
VAR_IN_OUT
	State : st_EthercatState;
END_VAR
State := InternalEtherCatState;
END_METHOD

END_FUNCTION_BLOCK

// ---- POUs/fbSafetyStateAndDiagDecode.TcPOU
FUNCTION_BLOCK fbSafetyStateAndDiagDecode
VAR_IN_OUT
		SafetyStatus :st_SafetyStatus;
END_VAR
VAR_INPUT 
		State :USINT;
		Diag  :USINT;
END_VAR

SafetyStatus.RawDiagCode:= Diag;
SafetyStatus.RawStateCode:=State;
SafetyStatus.State:=State;
SafetyStatus.FSoEMasterFailSafeActive:=Diag.7;
SafetyStatus.StartUp:= Diag.6;
SafetyStatus.FSoESlaveFailSafeActive:=Diag.5;
SafetyStatus.FSoESlaveError:=Diag.4;
SafetyStatus.Diagnosis:= SHL(Diag,4);

END_FUNCTION_BLOCK

// ---- POUs/fbStateMachineManager.TcPOU
FUNCTION_BLOCK fbStateMachineManager
VAR_INPUT
END_VAR
VAR_OUTPUT
END_VAR
VAR
	EthercatStateMachine : ARRAY[0..2] OF fbEthercatStateMachine[
									(EtherCatAddr:= '5.119.202.92.1.1',nSlaveAddr:=1001),
									(EtherCatAddr:= '5.119.202.92.1.1',nSlaveAddr:=1009),
									(EtherCatAddr:= '5.119.202.92.1.1',nSlaveAddr:=1006)];
									
	ModuleCount AT%I* : UINT;
	EtherCatStates: ARRAY[0..2] OF st_EthercatState;
END_VAR

FOR ModuleCount:= 0 TO 2 BY 1 DO 
EtherCatStateMachine[ModuleCount]();
EtherCatStateMachine[ModuleCount].GetState(State:= EtherCatStates[ModuleCount]);
EtherCatStates[ModuleCount].ModuleNumber:= UINT_TO_INT(ModuleCount);
END_FOR

END_FUNCTION_BLOCK

// ---- POUs/FB_SafeInfoState.TcPOU
FUNCTION_BLOCK FB_SafeInfoState
VAR
	State AT%I* :USINT;
	Diag AT%I* :USINT;
	Status :st_SafetyStatus;
	SafetyDecode : fbSafetyStateAndDiagDecode;
END_VAR

SafetyDecode(State:=State,Diag:=Diag,SafetyStatus:=Status);

END_FUNCTION_BLOCK

// ---- POUs/IDXMotor.TcPOU
   // function to house all commmands to do with idx motor 

FUNCTION_BLOCK IDXMotor IMPLEMENTS I_Motor
VAR_INPUT
	//
END_VAR
VAR_OUTPUT
END_VAR
VAR	

	Axis: AXIS_REF;
	//Enabled: BOOL := FALSE;
	Override: LREAL:=100;
	MotorError AT%I*	:WORD;
	MotorErrorSent : WORD;
	AxisErrorSent:UDINT;
	NCError : WORD;
	fbMessage : FB_TcMessage;
	EnableEventSent:BOOL:= TRUE;
	HomeEventSent:BOOL:=TRUE;
    fbAxisMoveAbsolute: MC_MoveAbsolute;	
	fbMcHome: MC_Home;
	fbAxisPower: MC_Power;
	fbReset: MC_Reset;
	fbMoveRel : MC_MoveRelative;
	MovementTarget : Lreal;
	MotorResetBit :REFERENCE TO USINT;
	
END_VAR

Axis.ReadStatus();

// cyclic events below 

IF NOT (MotorError = MotorErrorSent) THEN// Creates Event 
	MotorErrorSent:= MotorError;
	fbMessage.CreateEx(TC_Events.LinearMotor.IDXmotorError,0);
	fbMessage.ipArguments.Clear().AddDWord(MotorError);
	fbMessage.Send(0);
END_IF

IF NOT (Axis.NcToPlc.ErrorCode = AxisErrorSent) THEN// Creates Event 
	AxisErrorSent:= Axis.NcToPlc.ErrorCode;
	fbMessage.CreateEx(TC_Events.LinearMotor.AxisError,0);
	fbMessage.ipArguments.Clear().AddDWord(Axis.NcToPlc.ErrorCode);
	fbMessage.Send(0);
END_IF


METHOD PUBLIC Enable : BOOL
VAR_INPUT
EnableMotor :BOOL;
END_VAR



VAR
	PayloadPub: STRING :='Enabled';
	test: STRING;
	testlen: UDINT;
END_VAR
	fbAxisPower( // use in idx class
    Axis:= Axis,
    Enable:= EnableMotor,
    Enable_Positive:= EnableMotor,
    Enable_Negative:= EnableMotor,
    Override:= Override,
	Status=>Enable,
	Error=>
);
	

IF EnableMotor = EnableEventSent THEN	
	EnableEventSent := NOT EnableEventSent;
IF EnableMotor THEN
	fbMessage.CreateEx(TC_Events.LinearMotor.Motor_enabled,0);
ELSE
	fbMessage.CreateEx(TC_Events.LinearMotor.Motor_disabled,0);
END_IF
fbMessage.Send(0);
END_IF
fbMessage.RequestEventText(nLangId:=1033,sResult:=PayloadPub,nResultSize:=80);
END_METHOD

METHOD Estop : BOOL
VAR_INPUT
END_VAR
//stop motor mc stop
END_METHOD

METHOD FB_init : BOOL
VAR_INPUT
	bInitRetains : BOOL; // if TRUE, the retain variables are initialized (warm start / cold start)
	bInCopyCode : BOOL;  // if TRUE, the instance afterwards gets moved into the copy code (online change)
	ResetBit : REFERENCE TO USINT ;
	
END_VAR
//Axis :=AXIS_REF;
MotorResetBit REF= ResetBit;
fbMessage.CreateEx(TC_Events.LinearMotor.PLC_restarted,0);
	fbMessage.Send(0);
END_METHOD

METHOD PUBLIC Home : BOOL
VAR_IN_OUT
	Execute:BOOL;
END_VAR
VAR
	HomingDone:BOOL;
	HomingError:BOOL;
	HomingErrorID:UDINT;
END_VAR
// try changing limits to no error mode then home 


	fbMcHome(
	Axis:=Axis,
	Execute:=Execute,
	Position:=510,
	HomingMode:=MC_DefaultHoming,
	Busy=>Home,
	Done=>HomingDone,
	Error=> HomingError,
	ErrorID=> HomingErrorID
);
IF Home THEN
	Execute:= FALSE;
END_IF

IF Execute THEN
	HomeEventSent:= FALSE;
	fbMessage.CreateEx(TC_Events.LinearMotor.Homing,0);
	fbMessage.Send(0);
	//Execute:= FALSE;	
END_IF
IF HomingDone THEN
	fbMessage.CreateEx(TC_Events.LinearMotor.HomingComplete,0);
	fbMessage.Send(0);
END_IF

IF HomingError THEN
	Execute:= FALSE;
	fbMessage.CreateEx(TC_Events.LinearMotor.HomingFailed,0);
	fbMessage.ipArguments.Clear().AddDWord(HomingErrorID);
	fbMessage.Send(0);
END_IF
END_METHOD

METHOD PUBLIC Homed : BOOL
VAR_INPUT
END_VAR
Homed:=Axis.NcToPlc.StateDWord.1;
END_METHOD

METHOD MoveRelative : BOOL
VAR_INPUT
	Distance: LREAL;
	Velocity: LREAL;	
END_VAR
VAR_IN_OUT
	Execute: BOOL;
END_VAR
	fbMoveRel( // in idx class 
    Axis:= Axis,
    Execute:= Execute,
    Distance:= Distance,
    Velocity:= Velocity,);
	
		IF Execute THEN
	fbMessage.CreateEx(TC_Events.LinearMotor.RelativeMove,0);
	fbMessage.ipArguments.Clear();
	fbMessage.ipArguments.AddLReal(Distance);
	fbMessage.ipArguments.AddLReal(Velocity);
	fbMessage.Send(0);
	Execute := FALSE;
END_IF

IF fbMoveRel.Done  THEN
	fbMessage.CreateEx(TC_Events.LinearMotor.MoveComplete,0);
	fbMessage.Send(0);
	
END_IF
END_METHOD

METHOD MoveTo : BOOL
VAR_INPUT
	Position: LREAL;
	Velocity: LREAL;	
END_VAR

VAR_OUTPUT
	State: e_MCState;
	Target : LREAL;
	
END_VAR

VAR_IN_OUT
		Execute: BOOL;
END_VAR

VAR
	Done :BOOL;
	Busy:BOOL;
	Active:BOOL;
	Error:BOOL;
	CommandAborted : BOOL;
	
END_VAR
	fbAxisMoveAbsolute(  
    Axis:= Axis,
    Execute:= Execute,
    Position:= Position,
	BufferMode:= MC_BufferMode.MC_BlendingNext,
    Velocity:= Velocity,
	Done=> Done,
	Busy=>Busy,
	Active=> Active,
	Error=>Error,
	CommandAborted=>CommandAborted);
	
IF Done THEN
	State:= e_MCState.Done;
END_IF

IF Busy THEN
	State:= e_MCState.Busy;
END_IF

IF CommandAborted THEN
	State:= e_MCState.CommandAborted;
END_IF

IF Active THEN
	State:= e_MCState.Active;
END_IF
IF NOT Done AND NOT Busy AND NOT Active THEN
	State := e_MCState.Idle;
END_IF

IF Error THEN
	State:= e_MCState.Error;
END_IF
	
	IF Execute THEN
	MovementTarget := Position;
	fbMessage.CreateEx(TC_Events.LinearMotor.MotorMove,0);
	fbMessage.ipArguments.Clear();
	fbMessage.ipArguments.AddLReal(Position);
	fbMessage.ipArguments.AddLReal(Velocity);
	fbMessage.Send(0);
	Execute := FALSE;	
	END_IF

Target:= MovementTarget;

IF fbAxisMoveAbsolute.Done  THEN
	fbMessage.CreateEx(TC_Events.LinearMotor.MoveComplete,0);
	fbMessage.Send(0);


	
END_IF
END_METHOD

METHOD Position : LReal
VAR_INPUT
END_VAR
Position:= Axis.NcToPlc.ActPos;
END_METHOD

METHOD Reset : BOOL
VAR_IN_OUT
	ResetAxis:BOOL;
	//IDXControlByte1 :USINT;
END_VAR
fbReset(
Axis:=Axis,
Execute:=ResetAxis,
Done =>Reset);

IF resetAxis THEN
//IDXControlByte1 := 16#80;// restop linear Motor
MotorResetBit := 16#80;
fbMessage.CreateEx(TC_Events.LinearMotor.AxisReset,0);
fbMessage.send(0);
resetAxis := FALSE;
END_IF
END_METHOD

METHOD SetSpeed : BOOL
VAR_INPUT
END_VAR
END_METHOD

METHOD PUBLIC Status : ST_AxisStatus
VAR_INPUT
END_VAR
Status := Axis.Status;
END_METHOD

END_FUNCTION_BLOCK

// ---- POUs/fSafetyStateAndDiagDecode.TcPOU
FUNCTION fSafetyStateAndDiagDecode : st_SafetyStatus
VAR_INPUT
			State :USINT;
			Diag  :USINT;
		
END_VAR

fSafetyStateAndDiagDecode.RawDiagCode:= Diag;
fSafetyStateAndDiagDecode.RawStateCode:=State;
fSafetyStateAndDiagDecode.State:=State;
fSafetyStateAndDiagDecode.FSoEMasterFailSafeActive:=Diag.7;
fSafetyStateAndDiagDecode.StartUp:= Diag.6;
fSafetyStateAndDiagDecode.FSoESlaveFailSafeActive:=Diag.5;
fSafetyStateAndDiagDecode.FSoESlaveError:=Diag.4;
fSafetyStateAndDiagDecode.Diagnosis:= SHL(Diag,4);

END_FUNCTION

// ---- POUs/TestMode.TcPOU
FUNCTION_BLOCK PUBLIC TestMode
VAR_INPUT

END_VAR
VAR_OUTPUT
	TestingActive:BOOL;
END_VAR
VAR
	TestPosA: LREAL;
	TestPosB :LREAL;
	RefAxis : REFERENCE TO IDXMotor(); 
	AxisStatus : ST_AxisStatus;
	Operational :BOOL;
	InTargetPos: BOOL;
	HasJob :BOOL;
	DwellTimer: TON :=(PT:=T#5S,IN:=FALSE);
	Error :BOOL;// not used 
	TimerON: BOOL;
	Velo: LREAL;
	MoveExecute :BOOL;
	
END_VAR

//if testing active  can assume testing has begun 

//RefAxis.Status(Status =>AxisStatus); //problem
IF __ISVALIDREF(RefAxis) THEN 
	

AxisStatus := RefAxis.Status();
Operational:= AxisStatus.Operational;

IF TestingActive AND NOT Error THEN
	InTargetPos :=  AxisStatus.InTargetPosition;
	HasJob :=  AxisStatus.HasJob;
	
	IF Operational AND InTargetPos AND NOT HasJob THEN			
	 	TimerON:=TRUE;

	END_IF
	IF DwellTimer.Q THEN
		MoveExecute := TRUE;
		TimerON:=FALSE;
	END_IF

	IF ABS(RefAxis.Position()-TestPosA)<1 THEN
		RefAxis.MoveTo(Position:= TestPosB,Velocity:=Velo,Execute:=MoveExecute);
		ELSE
			RefAxis.MoveTo(Position:= TestPosA,Velocity:=Velo,Execute:=MoveExecute);
	END_IF

END_IF

IF NOT operational THEN
	TestingActive := FALSE;
END_IF

	

END_IF

DwellTimer(IN:=TimerON);

METHOD EndTest : BOOL
VAR_INPUT
	END :BOOL;
END_VAR
IF End THEN
	End:=FALSE;
	TestingActive:=FALSE;
END_IF
END_METHOD

METHOD StartTest : BOOL
VAR_INPUT
	PositionA: LREAL;
	PositionB :LREAL;
	Velocity : LREAL;
	Axis : REFERENCE TO IDXMotor();
	Dwell :TIME;
END_VAR
VAR_IN_OUT
	Execute :BOOL;
END_VAR
 IF Execute THEN
TestingActive :=TRUE;
TestPosA := PositionA;
TestPosB := PositionB;
Velo:= Velocity;
DwellTimer.PT := dwell;
RefAxis REF= Axis;
// error if not enabled 
RefAxis.MoveTo(Position:= TestPosA,Velocity:=Velocity,Execute:=Execute);
END_IF
END_METHOD

END_FUNCTION_BLOCK
